// TIA Portal V18 export
TYPE "MEStoPLC_MainCheckInStation1ST350_ext"
// stored: IsFailsafeCompliant false
   STRUCT
      PartTypeID : Int;   // 产品类型 1：11KW/2:22KW
      Station1PalletID : Int;   // 托盘号
      Station1PartSN : String[60];   // 产品主体码
      DataMatrixPartSN : String[60];   // 查询打标二维码
      Spare : Array[128..199] of Byte;   // 备用
      Massage : "MEStoPLC_AlarmMassage_ext";   // Process error code
   END_STRUCT;
END_TYPE
